TYPE Structure_Error :
STRUCT
	isError : BOOL := FALSE;
	errorMessage : STRING;
END_STRUCT
END_TYPE

(* stored: Version 1.1.0.1, ProductVersion 3.1.4024.12
   DUT Structure_Error: Id {55e2ca63-eaa5-4304-9730-bc68bea3f114} *)
